Staubli VAL3: min_.pgx

public program min_(num& x_nInput[], num& x_nResult)
  local num l_nElement
begin

  x_nResult = 99999
  for l_nElement = 0 to size(x_nInput)-1
    x_nResult = min(x_nResult, x_nInput[l_nElement])
  endFor

end
